// Mitsubishi GX Works2 project: SmartFarmModbusTempDx   PLC: FX3U/FX3UC

PROGRAM MAIN
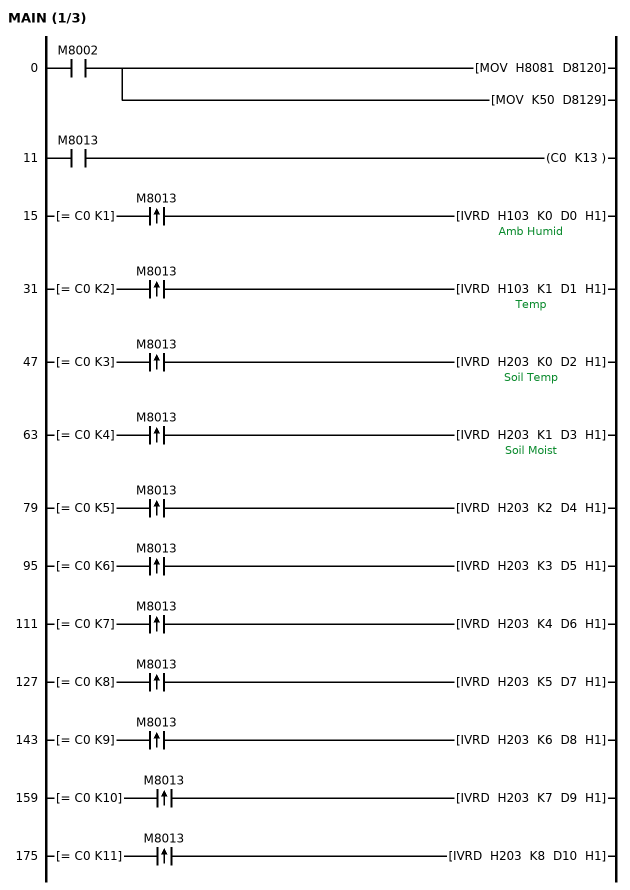
0     LD      M8002
      MOV     H8081 D8120
      MOV     K50 D8129
11    LD      M8013
      OUT     C0 K13
15    LD=     C0 K1
      ANDP    M8013
      IVRD    H103 K0 D0 H1  ; Amb Humid
31    LD=     C0 K2
      ANDP    M8013
      IVRD    H103 K1 D1 H1  ; Temp
47    LD=     C0 K3
      ANDP    M8013
      IVRD    H203 K0 D2 H1  ; Soil Temp
63    LD=     C0 K4
      ANDP    M8013
      IVRD    H203 K1 D3 H1  ; Soil Moist
79    LD=     C0 K5
      ANDP    M8013
      IVRD    H203 K2 D4 H1
95    LD=     C0 K6
      ANDP    M8013
      IVRD    H203 K3 D5 H1
111   LD=     C0 K7
      ANDP    M8013
      IVRD    H203 K4 D6 H1
127   LD=     C0 K8
      ANDP    M8013
      IVRD    H203 K5 D7 H1
143   LD=     C0 K9
      ANDP    M8013
      IVRD    H203 K6 D8 H1
159   LD=     C0 K10
      ANDP    M8013
      IVRD    H203 K7 D9 H1
175   LD=     C0 K11
      ANDP    M8013
      IVRD    H203 K8 D10 H1
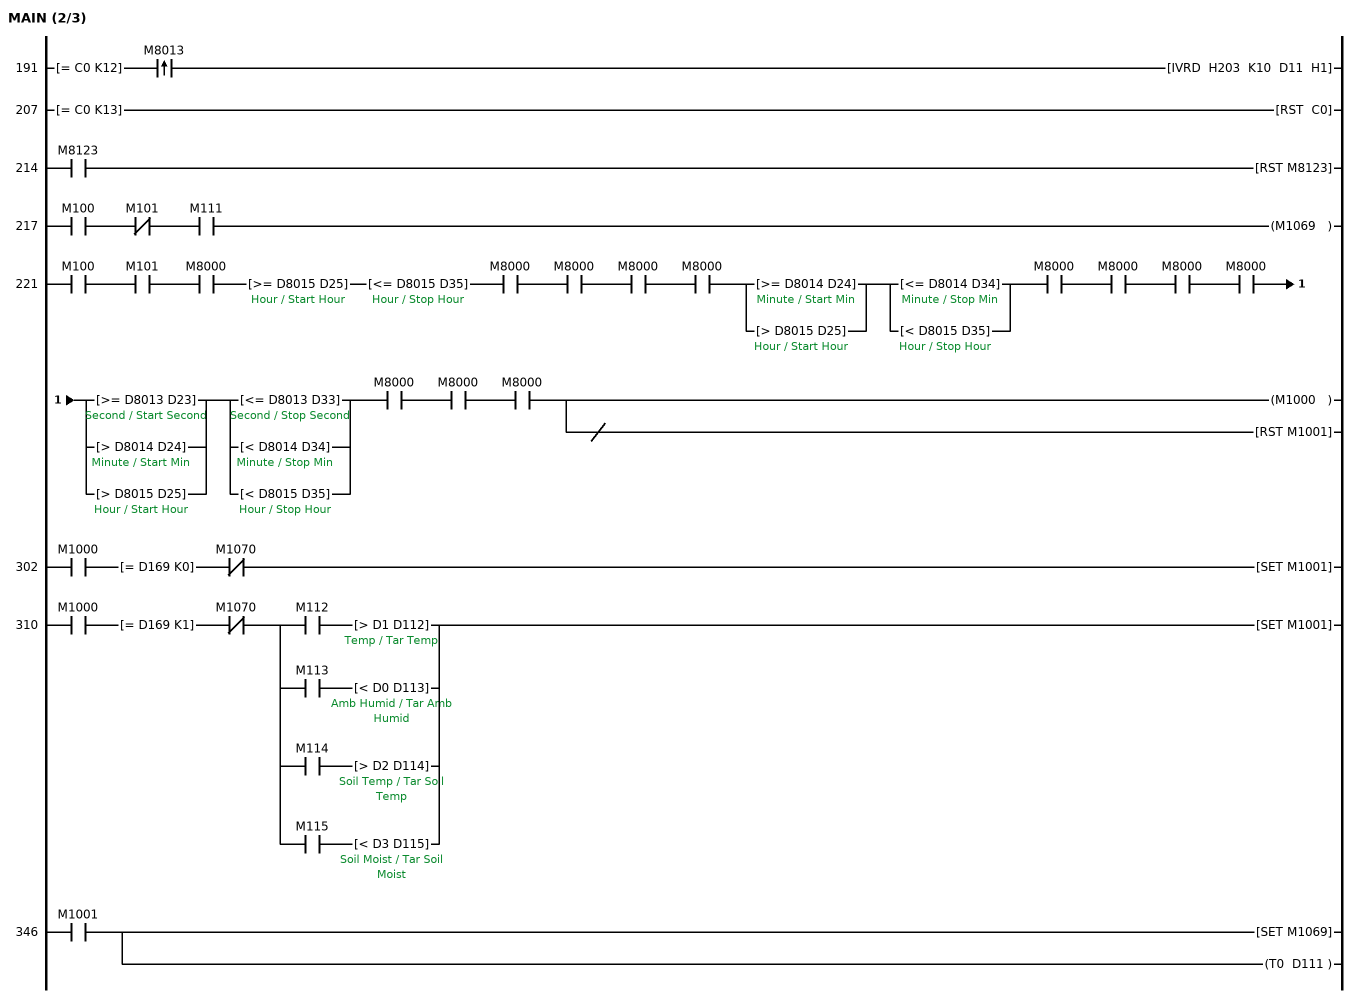
191   LD=     C0 K12
      ANDP    M8013
      IVRD    H203 K10 D11 H1
207   LD=     C0 K13
      RST     C0
214   LD      M8123
      RST     M8123
217   LD      M100
      ANI     M101
      AND     M111
      OUT     M1069
221   LD      M100
      AND     M101
      AND     M8000
      AND>=   D8015 D25  ; Hour / Start Hour
      AND<=   D8015 D35  ; Hour / Stop Hour
      AND     M8000
      AND     M8000
      AND     M8000
      AND     M8000
      LD>=    D8014 D24  ; Minute / Start Min
      OR>     D8015 D25  ; Hour / Start Hour
      ANB
      LD<=    D8014 D34  ; Minute / Stop Min
      OR<     D8015 D35  ; Hour / Stop Hour
      ANB
      AND     M8000
      AND     M8000
      AND     M8000
      AND     M8000
      LD>=    D8013 D23  ; Second / Start Second
      OR>     D8014 D24  ; Minute / Start Min
      OR>     D8015 D25  ; Hour / Start Hour
      ANB
      LD<=    D8013 D33  ; Second / Stop Second
      OR<     D8014 D34  ; Minute / Stop Min
      OR<     D8015 D35  ; Hour / Stop Hour
      ANB
      AND     M8000
      AND     M8000
      AND     M8000
      OUT     M1000
      INV
      RST     M1001
302   LD      M1000
      AND=    D169 K0
      ANI     M1070
      SET     M1001
310   LD      M1000
      AND=    D169 K1
      ANI     M1070
      LD      M112
      AND>    D1 D112  ; Temp / Tar Temp
      LD      M113
      AND<    D0 D113  ; Amb Humid / Tar Amb Humid
      ORB
      LD      M114
      AND>    D2 D114  ; Soil Temp / Tar Soil Temp
      ORB
      LD      M115
      AND<    D3 D115  ; Soil Moist / Tar Soil Moist
      ORB
      ANB
      SET     M1001
346   LD      M1001
      SET     M1069
      OUT     T0 D111
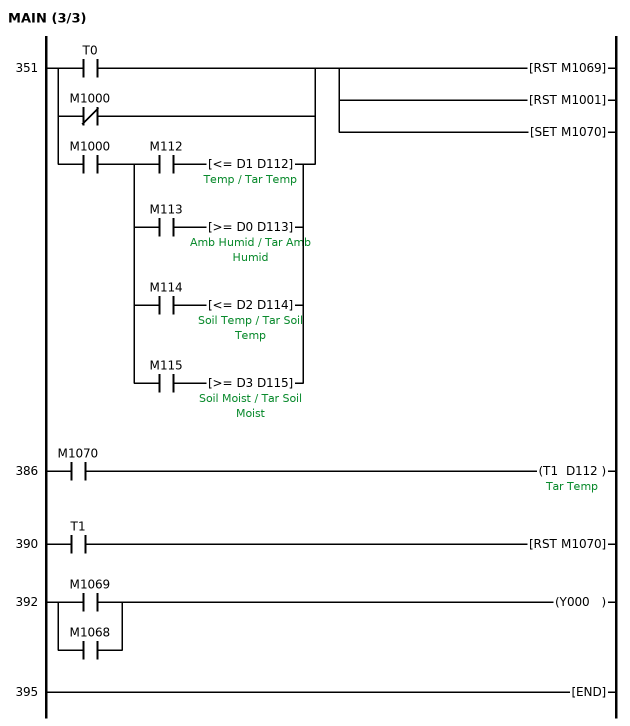
351   LD      T0
      ORI     M1000
      LD      M1000
      LD      M112
      AND<=   D1 D112  ; Temp / Tar Temp
      LD      M113
      AND>=   D0 D113  ; Amb Humid / Tar Amb Humid
      ORB
      LD      M114
      AND<=   D2 D114  ; Soil Temp / Tar Soil Temp
      ORB
      LD      M115
      AND>=   D3 D115  ; Soil Moist / Tar Soil Moist
      ORB
      ANB
      ORB
      RST     M1069
      RST     M1001
      SET     M1070
386   LD      M1070
      OUT     T1 D112  ; Tar Temp
390   LD      T1
      RST     M1070
392   LD      M1069
      OR      M1068
      OUT     Y000
395   END
END_PROGRAM
